// TIA Portal project "BottleWine" (V16)

(* hardware
DEVICE "S71500/ET200MP station_1"  S7-1500 station
   slot 0: "Rail_0"  Rack  6ES7 590-1***0-0AA0
   slot 1: "PLC_1"  CPU 1515-2 PN  6ES7 515-2AM00-0AB0  V1.8
      slot 3: "CPU display_1"  6ES7591-1BA00-0AA0
      slot 32768: "PROFINET interface_1"  X1
         slot 32769: "Port_1"  X1 P1
         slot 32770: "Port_2"  X1 P2
      slot 33024: "PROFINET interface_2"  X2
         slot 33025: "Port_1"  X2 P1
DEVICE "HMI_1"  TP1200 Comfort
   slot 0: "HMI_1"  TP1200 Comfort  6AV2 124-0MC01-0AX0  16.0.0.0
   slot 1: "HMI_RT_1"  TP1200 Comfort  6AV2 124-0MC01-0AX0  16.0.0.0
   slot 5: "HMI_1.IE_CP_1"  PROFINET Interface  16.0.0.0
      slot 1: "PROFINET Interface_1"  PROFINET Interface
         slot 1: "Port_1"  Port
         slot 2: "Port_2"  Port
   slot 7: "HMI_1.MPI/DP_CP_1"  MPI/DP Interface  16.0.0.0
*)

// ===== PLC "PLC_1"  CPU 1515-2 PN =====

VAR_GLOBAL   // PLC tag table "Default tag table"
   "P_TRIG1" AT %M5.1 : Bool;
   "Start" AT %M0.0 : Bool;
   "Production_Line" AT %M0.1 : Bool;
   "WhiteBottleSensor" AT %M0.2 : Bool;
   "P_TRIG2" AT %M5.2 : Bool;
   "FillWhiteWine" AT %M0.3 : Bool;
   "WhiteBottle" AT %M0.4 : Bool;
   "DarkBootle" AT %M0.5 : Bool;
   "P_TRIG3" AT %M5.3 : Bool;
   "DarkBottleSensor" AT %M0.6 : Bool;
   "P_TRIG4" AT %M0.7 : Bool;
   "FillDarkWine" AT %M1.0 : Bool;
   "fillingWhite" AT %M1.1 : Bool;
   "fillingDark" AT %M1.2 : Bool;
   "P_TRIG5" AT %M1.3 : Bool;
   "filling" AT %M1.4 : Bool;
   "filling1" AT %M1.5 : Bool;
   "filling2" AT %M1.6 : Bool;
   "PTRIG_6" AT %M1.7 : Bool;
   "Corking" AT %M2.0 : Bool;
   "P_TRIG6" AT %M2.1 : Bool;
   "P_TRIG7" AT %M2.2 : Bool;
   "Corking Sensor" AT %M2.3 : Bool;
   "P_TRIG8" AT %M2.4 : Bool;
   "label" AT %M2.5 : Bool;
   "P_TRIG9" AT %M2.6 : Bool;
   "label Sensor" AT %M2.7 : Bool;
   "P_TRIG10" AT %M3.0 : Bool;
   "NeckLabel Sensor" AT %M3.1 : Bool;
   "P_TRIG11" AT %M3.2 : Bool;
   "NecklabelWhite" AT %M3.3 : Bool;
   "P_TRIG12" AT %M3.4 : Bool;
   "corking1" AT %M3.5 : Bool;
   "corking2" AT %M3.6 : Bool;
   "Corking White Wine" AT %M3.7 : Bool;
   "Corking Dark Wine" AT %M4.0 : Bool;
   "cukubik" AT %M4.1 : Bool;
END_VAR

ORGANIZATION_BLOCK "Main"   // OB1, LAD, ProgramCycle
TITLE = "Main Program Sweep (Cycle)"
{ S7_Optimized_Access := 'TRUE' }
VERSION : 0.1
   VAR_INPUT
      Initial_Call : Bool;   // Initial call of this OB
      Remanence : Bool;   // =True, if remanent data are available
   END_VAR
   VAR_TEMP   // added for the SCL form of the ladder/FBD networks
      _w1 : Bool;
      _w2 : Bool;
      _w3 : Bool;
      _w4 : Bool;
   END_VAR
BEGIN

REGION Network 1
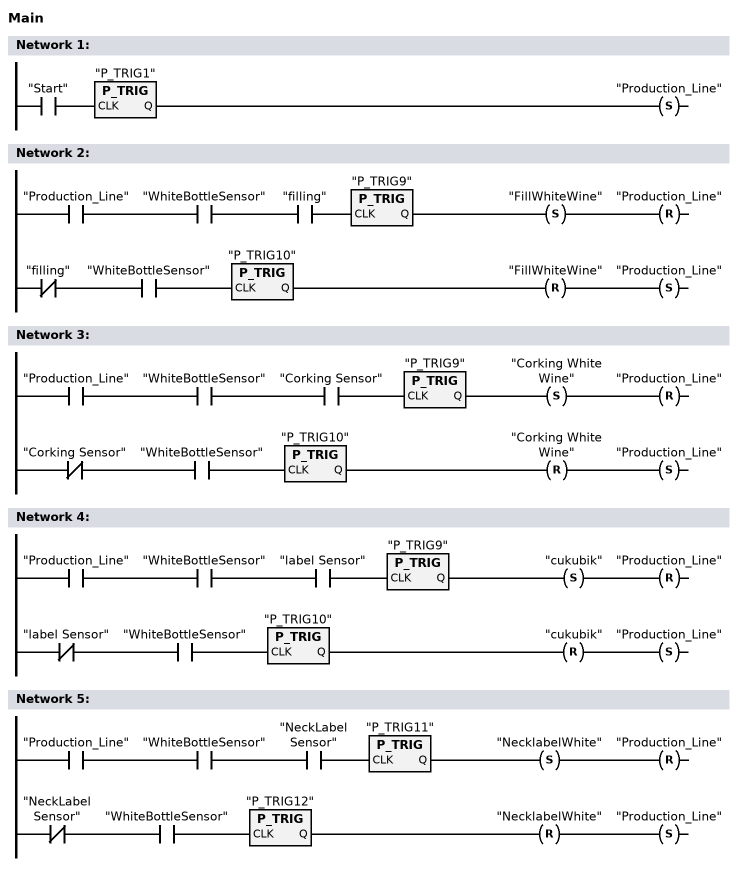
   RUNG wire#powerrail
      Contact( "Start" )
      P_Trig( "P_TRIG1" )
      S_Coil( "Production_Line" )
   END_RUNG
   // the same network as SCL:
   #_w1 := "Start" AND NOT "P_TRIG1";   // rising edge
   "P_TRIG1" := "Start";
   IF #_w1 THEN "Production_Line" := TRUE; END_IF;
END_REGION

REGION Network 2
   RUNG wire#powerrail
      Contact( "Production_Line" )
      Contact( "WhiteBottleSensor" )
      Contact( "filling" )
      P_Trig( "P_TRIG9" )
      S_Coil( "FillWhiteWine" )
      R_Coil( "Production_Line" )
   END_RUNG
   RUNG wire#powerrail
      I_Contact( "filling" )
      Contact( "WhiteBottleSensor" )
      P_Trig( "P_TRIG10" )
      R_Coil( "FillWhiteWine" )
      S_Coil( "Production_Line" )
   END_RUNG
   // the same network as SCL:
   #_w1 := "Production_Line" AND "WhiteBottleSensor" AND "filling";
   #_w2 := #_w1 AND NOT "P_TRIG9";   // rising edge
   "P_TRIG9" := #_w1;
   IF #_w2 THEN
       "FillWhiteWine" := TRUE;
       "Production_Line" := FALSE;
   END_IF;
   #_w3 := NOT "filling" AND "WhiteBottleSensor";
   #_w4 := #_w3 AND NOT "P_TRIG10";   // rising edge
   "P_TRIG10" := #_w3;
   IF #_w4 THEN
       "FillWhiteWine" := FALSE;
       "Production_Line" := TRUE;
   END_IF;
END_REGION

REGION Network 3
   RUNG wire#powerrail
      Contact( "Production_Line" )
      Contact( "WhiteBottleSensor" )
      Contact( "Corking Sensor" )
      P_Trig( "P_TRIG9" )
      S_Coil( "Corking White Wine" )
      R_Coil( "Production_Line" )
   END_RUNG
   RUNG wire#powerrail
      I_Contact( "Corking Sensor" )
      Contact( "WhiteBottleSensor" )
      P_Trig( "P_TRIG10" )
      R_Coil( "Corking White Wine" )
      S_Coil( "Production_Line" )
   END_RUNG
   // the same network as SCL:
   #_w1 := "Production_Line" AND "WhiteBottleSensor" AND "Corking Sensor";
   #_w2 := #_w1 AND NOT "P_TRIG9";   // rising edge
   "P_TRIG9" := #_w1;
   IF #_w2 THEN
       "Corking White Wine" := TRUE;
       "Production_Line" := FALSE;
   END_IF;
   #_w3 := NOT "Corking Sensor" AND "WhiteBottleSensor";
   #_w4 := #_w3 AND NOT "P_TRIG10";   // rising edge
   "P_TRIG10" := #_w3;
   IF #_w4 THEN
       "Corking White Wine" := FALSE;
       "Production_Line" := TRUE;
   END_IF;
END_REGION

REGION Network 4
   RUNG wire#powerrail
      Contact( "Production_Line" )
      Contact( "WhiteBottleSensor" )
      Contact( "label Sensor" )
      P_Trig( "P_TRIG9" )
      S_Coil( "cukubik" )
      R_Coil( "Production_Line" )
   END_RUNG
   RUNG wire#powerrail
      I_Contact( "label Sensor" )
      Contact( "WhiteBottleSensor" )
      P_Trig( "P_TRIG10" )
      R_Coil( "cukubik" )
      S_Coil( "Production_Line" )
   END_RUNG
   // the same network as SCL:
   #_w1 := "Production_Line" AND "WhiteBottleSensor" AND "label Sensor";
   #_w2 := #_w1 AND NOT "P_TRIG9";   // rising edge
   "P_TRIG9" := #_w1;
   IF #_w2 THEN
       "cukubik" := TRUE;
       "Production_Line" := FALSE;
   END_IF;
   #_w3 := NOT "label Sensor" AND "WhiteBottleSensor";
   #_w4 := #_w3 AND NOT "P_TRIG10";   // rising edge
   "P_TRIG10" := #_w3;
   IF #_w4 THEN
       "cukubik" := FALSE;
       "Production_Line" := TRUE;
   END_IF;
END_REGION

REGION Network 5
   RUNG wire#powerrail
      Contact( "Production_Line" )
      Contact( "WhiteBottleSensor" )
      Contact( "NeckLabel Sensor" )
      P_Trig( "P_TRIG11" )
      S_Coil( "NecklabelWhite" )
      R_Coil( "Production_Line" )
   END_RUNG
   RUNG wire#powerrail
      I_Contact( "NeckLabel Sensor" )
      Contact( "WhiteBottleSensor" )
      P_Trig( "P_TRIG12" )
      R_Coil( "NecklabelWhite" )
      S_Coil( "Production_Line" )
   END_RUNG
   // the same network as SCL:
   #_w1 := "Production_Line" AND "WhiteBottleSensor" AND "NeckLabel Sensor";
   #_w2 := #_w1 AND NOT "P_TRIG11";   // rising edge
   "P_TRIG11" := #_w1;
   IF #_w2 THEN
       "NecklabelWhite" := TRUE;
       "Production_Line" := FALSE;
   END_IF;
   #_w3 := NOT "NeckLabel Sensor" AND "WhiteBottleSensor";
   #_w4 := #_w3 AND NOT "P_TRIG12";   // rising edge
   "P_TRIG12" := #_w3;
   IF #_w4 THEN
       "NecklabelWhite" := FALSE;
       "Production_Line" := TRUE;
   END_IF;
END_REGION
END_ORGANIZATION_BLOCK

(* ===== HMI "HMI_RT_1" =====
system functions are stored by id; their names below are inferred from use
connection "HMI_Connection_1": ETHERNET, S7_1500_OMS

HMI tags "Default tag table"
   "Tag_ScreenNumber" : UInt, internal
   "Start" : Bool = PLC Start AT %M0.0, 1 s
   "Production_Line" : Bool = PLC Production_Line AT %M0.1, 1 s
   "WhiteBottle" : Bool = PLC WhiteBottle AT %M0.4, 1 s
   "DarkBootle" : Bool = PLC DarkBootle AT %M0.5, 1 s
   "filling" : Bool = PLC filling AT %M1.4, 1 s
   "FillWhiteWine" : Bool = PLC FillWhiteWine AT %M0.3, 1 s
   "WhiteBottleSensor" : Bool = PLC WhiteBottleSensor AT %M0.2, 1 s
   "DarkBottleSensor" : Bool = PLC DarkBottleSensor AT %M0.6, 1 s
   "FillDarkWine" : Bool = PLC FillDarkWine AT %M1.0, 1 s
   "Corking Sensor" : Bool = PLC "Corking Sensor" AT %M2.3, 1 s
   "Corking" : Bool = PLC Corking AT %M2.0, 1 s
   "label Sensor" : Bool = PLC "label Sensor" AT %M2.7, 1 s
   "label" : Bool = PLC label AT %M2.5, 1 s
   "NeckLabel Sensor" : Bool = PLC "NeckLabel Sensor" AT %M3.1, 1 s
   "NecklabelWhite" : Bool = PLC NecklabelWhite AT %M3.3, 1 s
   "Corking White Wine" : Bool = PLC "Corking White Wine" AT %M3.7, 1 s
   "Corking Dark Wine" : Bool = PLC "Corking Dark Wine" AT %M4.0, 1 s
   "cukubik" : Bool = PLC cukubik AT %M4.1, 1 s

screen "Root screen" 1280x740, template "Template_1"
   on GenerateScreen: SetTag("Tag_ScreenNumber", 1)
   Button "Button_1" at 75,71 size 96x32; TextOff 'Start'
      on Press: InvertBit("Start")
   Circle "Circle_1" at 229,61 size 48x48
      Appearance <- "Start"
   TextField "Text field_1" at 25,136 size 155x25; Text 'Production Line'
   Circle "Circle_2" at 229,118 size 48x48
      Appearance <- "Production_Line"
   Button "Button_2" at 27,184 size 179x32; TextOff 'White Bottle Sensor'
      on Press: InvertBit("WhiteBottleSensor")
   Circle "Circle_3" at 230,174 size 48x48
      Appearance <- "WhiteBottleSensor"
   Button "Button_3" at 29,241 size 176x32; TextOff 'Dark Bottle Sensor'
      Appearance <- "DarkBootle"
      on Press: InvertBit("DarkBottleSensor")
   Circle "Circle_4" at 230,232 size 48x48
      Appearance <- "DarkBottleSensor"
   Button "Button_4" at 29,297 size 96x32; TextOff 'Filling'
      on Press: InvertBit("filling")
   Circle "Circle_5" at 230,294 size 48x48
      Appearance <- "filling"
   TextField "Text field_2" at 415,71 size 148x25; Text 'Fill White Wine'
   Circle "Circle_6" at 585,55 size 48x48
      Appearance <- "FillWhiteWine"
   Button "Button_5" at 30,377 size 184x32; TextOff 'Corking Sensor'
      on Press: InvertBit("Corking Sensor")
   Circle "Circle_8" at 237,360 size 48x48
      Appearance <- "Corking Sensor"
   TextField "Text field_4" at 406,185 size 139x25; Text 'Corking White'
   Circle "Circle_9" at 585,168 size 48x48
      Appearance <- "Corking White Wine"
   Button "Button_6" at 25,446 size 165x32; TextOff 'Label Sensor'
      on Press: InvertBit("label Sensor")
   Circle "Circle_10" at 237,434 size 48x48
      Appearance <- "label Sensor"
   TextField "Text field_5" at 406,241 size 170x25; Text 'Label White Wine'
   Circle "Circle_11" at 585,227 size 48x48
      Appearance <- "cukubik"
   TextField "Text field_6" at 347,307 size 222x25; Text 'Neck Label White Wine'
   Circle "Circle_12" at 585,283 size 48x48
      Appearance <- "NecklabelWhite"
   Button "Button_7" at 30,514 size 157x32; TextOff 'Neck Label Sensor'
      on Press: InvertBit("NeckLabel Sensor")
   Circle "Circle_13" at 235,504 size 48x48
      Appearance <- "NeckLabel Sensor"

Template "Template_1" 1280x740
   Button "Exit" at 1200,679 size 78x59; TextOff 'Exit'; PictureOff "ExitRuntime_TP1200_Comfort_TR"; PictureOn "ExitRuntime_TP1200_Comfort_TR"
      on Release: StopRuntime(0)
   Button "Template_Button" at 1120,679 size 78x59; TextOff 'Text'
   Button "Template_Button_1" at 1040,679 size 78x59; TextOff 'Text'
   Button "Template_Button_2" at 960,679 size 78x59; TextOff 'Text'
   Button "Template_Button_3" at 880,679 size 78x59; TextOff 'Text'
   Button "Template_Button_4" at 800,679 size 78x59; TextOff 'Text'
   Button "Template_Button_5" at 720,679 size 78x59; TextOff 'Text'
   Button "Template_Button_6" at 640,679 size 78x59; TextOff 'Text'
   Button "Template_Button_7" at 561,679 size 78x59; TextOff 'Text'
   Button "Template_Button_8" at 481,679 size 78x59; TextOff 'Text'
   Button "Template_Button_9" at 401,679 size 78x59; TextOff 'Text'
   Button "Template_Button_10" at 321,679 size 78x59; TextOff 'Text'
   Button "Template_Button_11" at 241,679 size 78x59; TextOff 'Text'
   Button "Template_Button_12" at 161,679 size 78x59; TextOff 'Text'
   Button "Template_Button_13" at 81,679 size 78x59; TextOff 'Text'
   Button "Start screen" at 1,679 size 78x59; TextOff 'Start screen'; PictureOff "NavigateHome_TP1200_Comfort_TR"; PictureOn "NavigateHome_TP1200_Comfort_TR"
      on Release: ActivateScreen("Root screen", 0)
*)